FUNCTION_BLOCK Fb_Motion
VAR_INPUT
END_VAR
VAR_OUTPUT
END_VAR
VAR
	
	MCPower: MC_Power;
	McStop: MC_Stop;
	MCMoveAbs: MC_MoveAbsolute;
	McReset: MC_Reset;
	
END_VAR
VAR_IN_OUT
	
	Axis : AXIS_REF;
	staxisinterface : stAxisInterface;

END_VAR

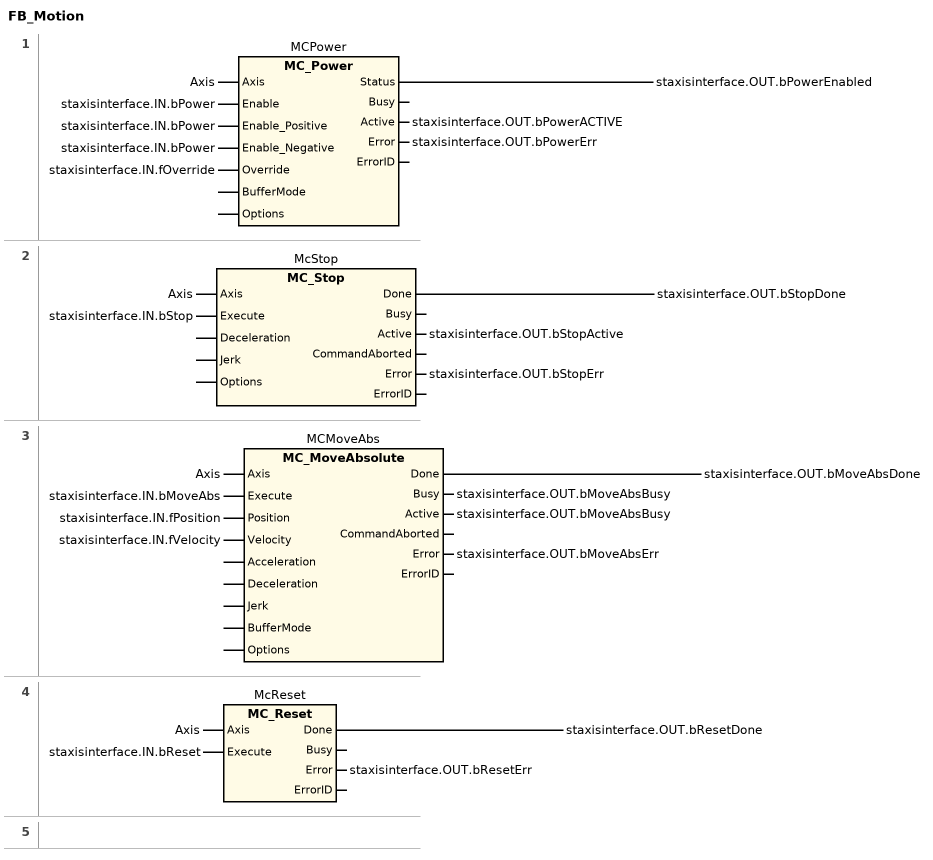
// NETWORK 1
MCPower(
    Axis := Axis,
    Enable := staxisinterface.IN.bPower,
    Enable_Positive := staxisinterface.IN.bPower,
    Enable_Negative := staxisinterface.IN.bPower,
    Override := staxisinterface.IN.fOverride,
    Active => staxisinterface.OUT.bPowerACTIVE,
    Error => staxisinterface.OUT.bPowerErr); // MC_Power
staxisinterface.OUT.bPowerEnabled := MCPower.Status;

// NETWORK 2
McStop(
    Axis := Axis,
    Execute := staxisinterface.IN.bStop,
    Active => staxisinterface.OUT.bStopActive,
    Error => staxisinterface.OUT.bStopErr); // MC_Stop
staxisinterface.OUT.bStopDone := McStop.Done;

// NETWORK 3
MCMoveAbs(
    Axis := Axis,
    Execute := staxisinterface.IN.bMoveAbs,
    Position := staxisinterface.IN.fPosition,
    Velocity := staxisinterface.IN.fVelocity,
    Busy => staxisinterface.OUT.bMoveAbsBusy,
    Active => staxisinterface.OUT.bMoveAbsBusy,
    Error => staxisinterface.OUT.bMoveAbsErr); // MC_MoveAbsolute
staxisinterface.OUT.bMoveAbsDone := MCMoveAbs.Done;

// NETWORK 4
McReset(Axis := Axis, Execute := staxisinterface.IN.bReset, Error => staxisinterface.OUT.bResetErr); // MC_Reset
staxisinterface.OUT.bResetDone := McReset.Done;

// NETWORK 5

END_FUNCTION_BLOCK

(* stored: Version 1.1.0.1, ProductVersion 3.1.4024.4
   POU FB_Motion: Id {c7306cfe-b94d-4239-af91-e0803bc4e3f3}, SpecialFunc None *)
